(* Logix 5000 project; controller BTS01 vendor 1 type 14 code 217 rev 32.14; software revision 32.04; part 10 of 15 *)
(* tags used below, declared in another part *)
   Alarm_Active : DINT;
   Alarm_TMR : TIMER[17,32];
   ALM_ENABLE : DINT[25];
   GlobalAlmAck : BOOL;
   HMI_Alarms_Active : BOOL;
   HMI_Global_Alarm_Ack_PB : BOOL;
   HMIAlarms : DINT[25];   // Alarm Trigger Array
   HMIAlarmsMsg : STRING64[17,32];   // Alarm Descriptions to Match Alarm Trigger Array
(* Alarm, continued *)

ROUTINE Alarm_10   (* ladder *)
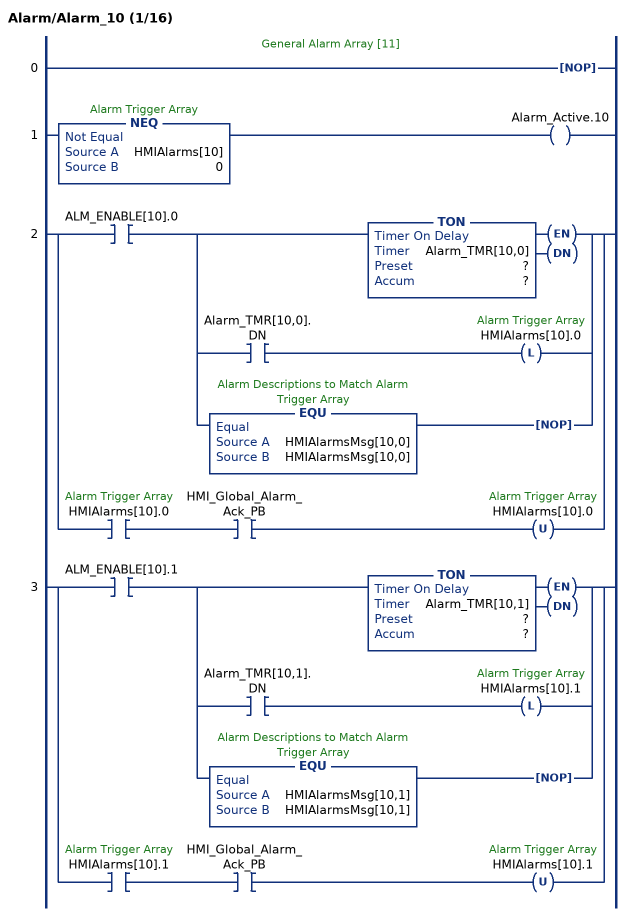
   // General Alarm Array [11]
   0: NOP();
   1: NEQ(HMIAlarms[10],0)OTE(Alarm_Active.10);
   2: [XIC(ALM_ENABLE[10].0) [TON(Alarm_TMR[10,0],?,?) ,XIC(Alarm_TMR[10,0].DN) OTL(HMIAlarms[10].0) ,EQU(HMIAlarmsMsg[10,0],HMIAlarmsMsg[10,0]) NOP() ] ,XIC(HMIAlarms[10].0) XIC(HMI_Global_Alarm_Ack_PB) OTU(HMIAlarms[10].0) ];
   3: [XIC(ALM_ENABLE[10].1) [TON(Alarm_TMR[10,1],?,?) ,XIC(Alarm_TMR[10,1].DN) OTL(HMIAlarms[10].1) ,EQU(HMIAlarmsMsg[10,1],HMIAlarmsMsg[10,1]) NOP() ] ,XIC(HMIAlarms[10].1) XIC(HMI_Global_Alarm_Ack_PB) OTU(HMIAlarms[10].1) ];
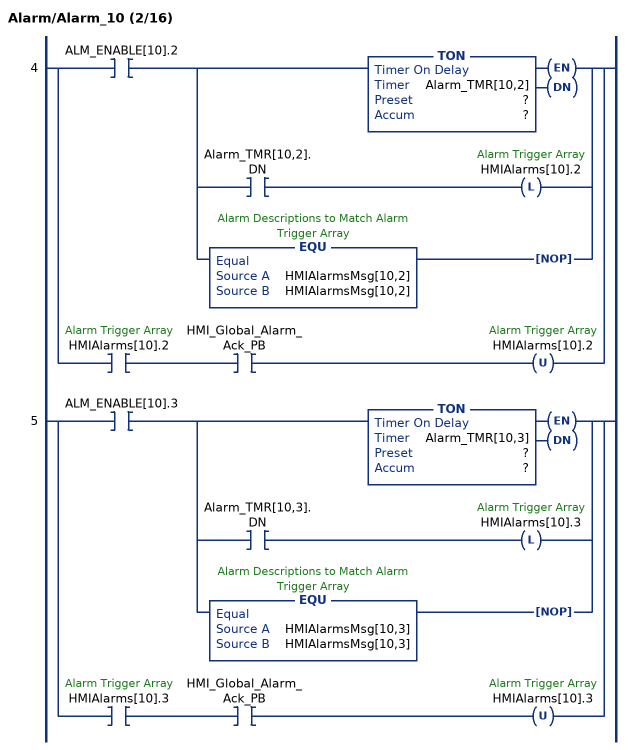
   4: [XIC(ALM_ENABLE[10].2) [TON(Alarm_TMR[10,2],?,?) ,XIC(Alarm_TMR[10,2].DN) OTL(HMIAlarms[10].2) ,EQU(HMIAlarmsMsg[10,2],HMIAlarmsMsg[10,2]) NOP() ] ,XIC(HMIAlarms[10].2) XIC(HMI_Global_Alarm_Ack_PB) OTU(HMIAlarms[10].2) ];
   5: [XIC(ALM_ENABLE[10].3) [TON(Alarm_TMR[10,3],?,?) ,XIC(Alarm_TMR[10,3].DN) OTL(HMIAlarms[10].3) ,EQU(HMIAlarmsMsg[10,3],HMIAlarmsMsg[10,3]) NOP() ] ,XIC(HMIAlarms[10].3) XIC(HMI_Global_Alarm_Ack_PB) OTU(HMIAlarms[10].3) ];
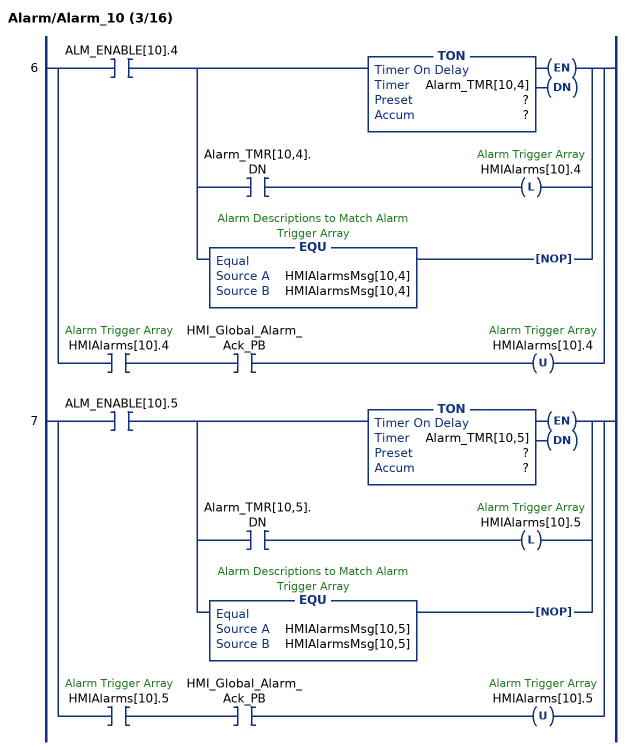
   6: [XIC(ALM_ENABLE[10].4) [TON(Alarm_TMR[10,4],?,?) ,XIC(Alarm_TMR[10,4].DN) OTL(HMIAlarms[10].4) ,EQU(HMIAlarmsMsg[10,4],HMIAlarmsMsg[10,4]) NOP() ] ,XIC(HMIAlarms[10].4) XIC(HMI_Global_Alarm_Ack_PB) OTU(HMIAlarms[10].4) ];
   7: [XIC(ALM_ENABLE[10].5) [TON(Alarm_TMR[10,5],?,?) ,XIC(Alarm_TMR[10,5].DN) OTL(HMIAlarms[10].5) ,EQU(HMIAlarmsMsg[10,5],HMIAlarmsMsg[10,5]) NOP() ] ,XIC(HMIAlarms[10].5) XIC(HMI_Global_Alarm_Ack_PB) OTU(HMIAlarms[10].5) ];
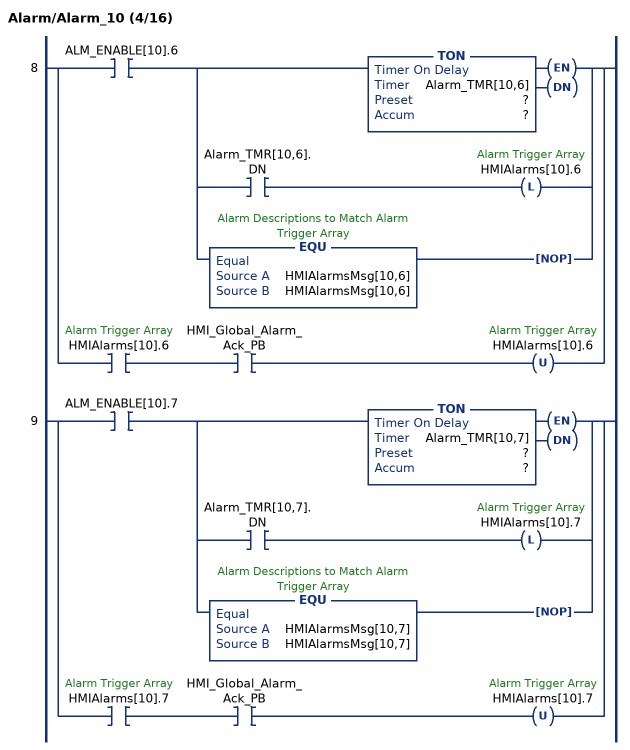
   8: [XIC(ALM_ENABLE[10].6) [TON(Alarm_TMR[10,6],?,?) ,XIC(Alarm_TMR[10,6].DN) OTL(HMIAlarms[10].6) ,EQU(HMIAlarmsMsg[10,6],HMIAlarmsMsg[10,6]) NOP() ] ,XIC(HMIAlarms[10].6) XIC(HMI_Global_Alarm_Ack_PB) OTU(HMIAlarms[10].6) ];
   9: [XIC(ALM_ENABLE[10].7) [TON(Alarm_TMR[10,7],?,?) ,XIC(Alarm_TMR[10,7].DN) OTL(HMIAlarms[10].7) ,EQU(HMIAlarmsMsg[10,7],HMIAlarmsMsg[10,7]) NOP() ] ,XIC(HMIAlarms[10].7) XIC(HMI_Global_Alarm_Ack_PB) OTU(HMIAlarms[10].7) ];
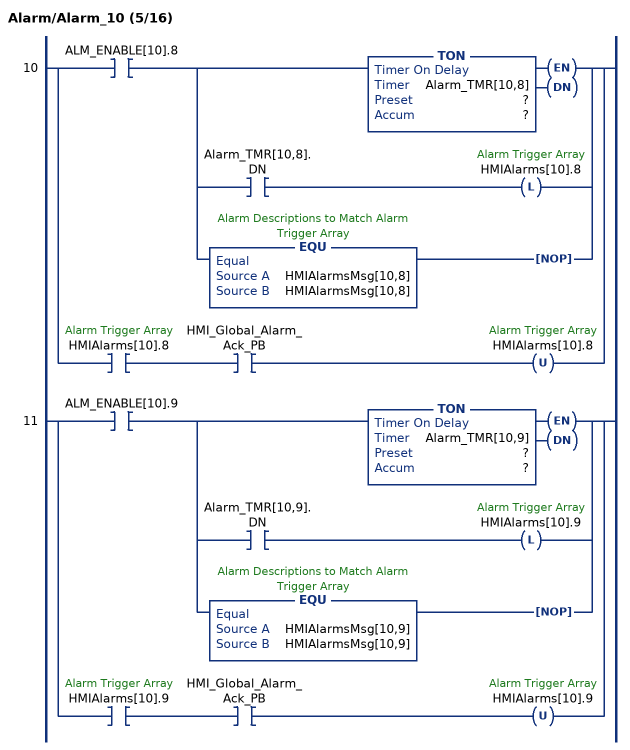
   10: [XIC(ALM_ENABLE[10].8) [TON(Alarm_TMR[10,8],?,?) ,XIC(Alarm_TMR[10,8].DN) OTL(HMIAlarms[10].8) ,EQU(HMIAlarmsMsg[10,8],HMIAlarmsMsg[10,8]) NOP() ] ,XIC(HMIAlarms[10].8) XIC(HMI_Global_Alarm_Ack_PB) OTU(HMIAlarms[10].8) ];
   11: [XIC(ALM_ENABLE[10].9) [TON(Alarm_TMR[10,9],?,?) ,XIC(Alarm_TMR[10,9].DN) OTL(HMIAlarms[10].9) ,EQU(HMIAlarmsMsg[10,9],HMIAlarmsMsg[10,9]) NOP() ] ,XIC(HMIAlarms[10].9) XIC(HMI_Global_Alarm_Ack_PB) OTU(HMIAlarms[10].9) ];
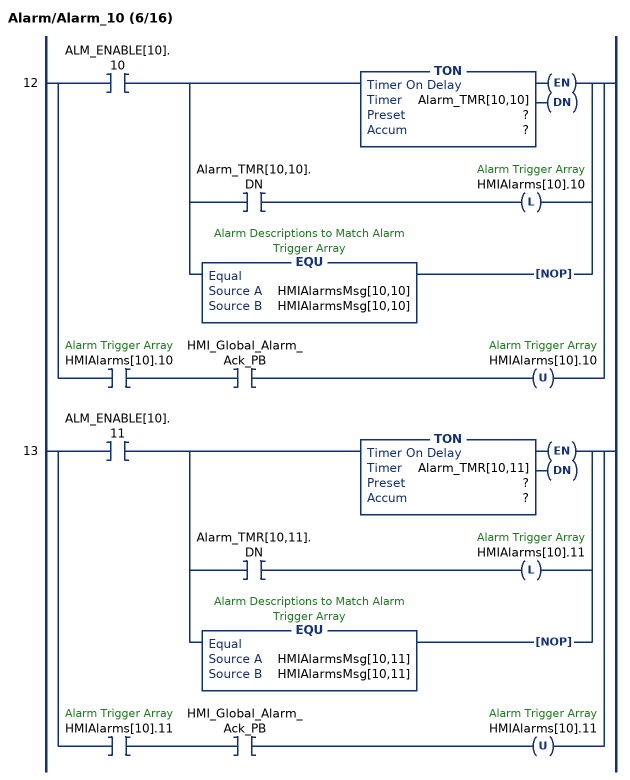
   12: [XIC(ALM_ENABLE[10].10) [TON(Alarm_TMR[10,10],?,?) ,XIC(Alarm_TMR[10,10].DN) OTL(HMIAlarms[10].10) ,EQU(HMIAlarmsMsg[10,10],HMIAlarmsMsg[10,10]) NOP() ] ,XIC(HMIAlarms[10].10) XIC(HMI_Global_Alarm_Ack_PB) OTU(HMIAlarms[10].10) ];
   13: [XIC(ALM_ENABLE[10].11) [TON(Alarm_TMR[10,11],?,?) ,XIC(Alarm_TMR[10,11].DN) OTL(HMIAlarms[10].11) ,EQU(HMIAlarmsMsg[10,11],HMIAlarmsMsg[10,11]) NOP() ] ,XIC(HMIAlarms[10].11) XIC(HMI_Global_Alarm_Ack_PB) OTU(HMIAlarms[10].11) ];
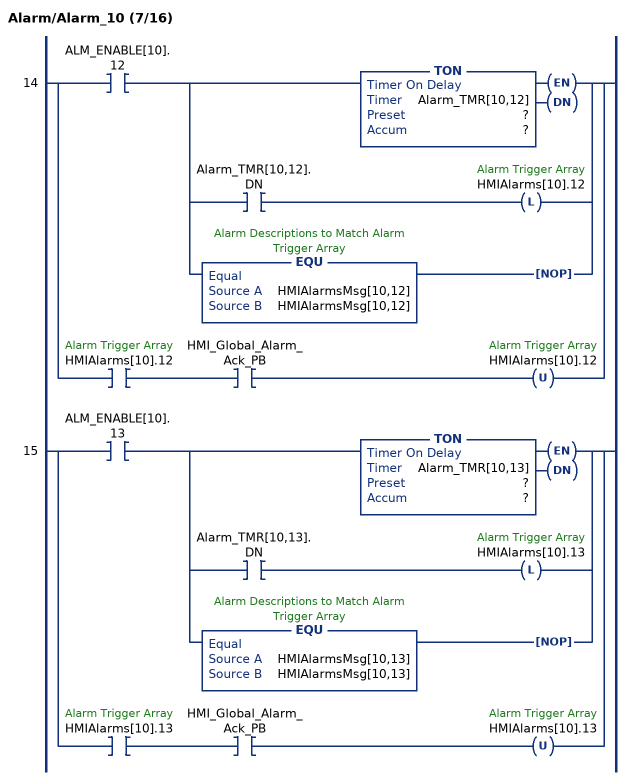
   14: [XIC(ALM_ENABLE[10].12) [TON(Alarm_TMR[10,12],?,?) ,XIC(Alarm_TMR[10,12].DN) OTL(HMIAlarms[10].12) ,EQU(HMIAlarmsMsg[10,12],HMIAlarmsMsg[10,12]) NOP() ] ,XIC(HMIAlarms[10].12) XIC(HMI_Global_Alarm_Ack_PB) OTU(HMIAlarms[10].12) ];
   15: [XIC(ALM_ENABLE[10].13) [TON(Alarm_TMR[10,13],?,?) ,XIC(Alarm_TMR[10,13].DN) OTL(HMIAlarms[10].13) ,EQU(HMIAlarmsMsg[10,13],HMIAlarmsMsg[10,13]) NOP() ] ,XIC(HMIAlarms[10].13) XIC(HMI_Global_Alarm_Ack_PB) OTU(HMIAlarms[10].13) ];
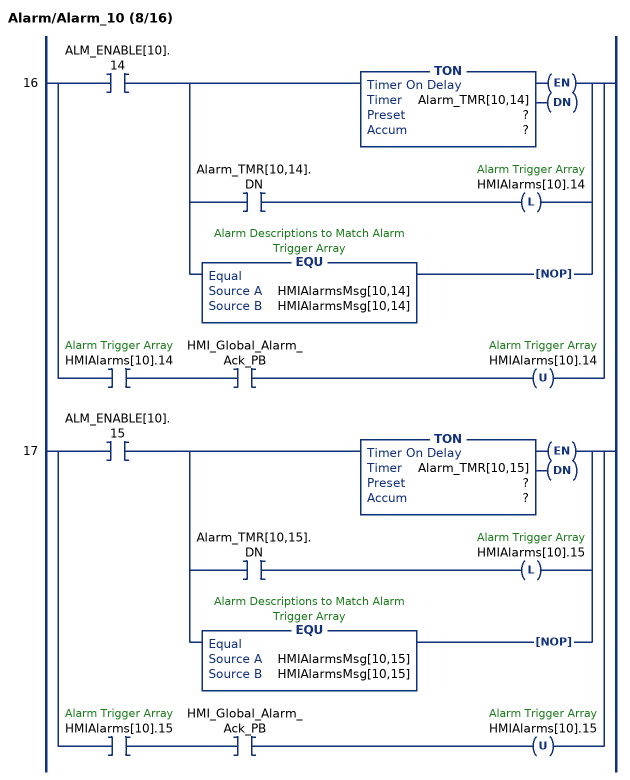
   16: [XIC(ALM_ENABLE[10].14) [TON(Alarm_TMR[10,14],?,?) ,XIC(Alarm_TMR[10,14].DN) OTL(HMIAlarms[10].14) ,EQU(HMIAlarmsMsg[10,14],HMIAlarmsMsg[10,14]) NOP() ] ,XIC(HMIAlarms[10].14) XIC(HMI_Global_Alarm_Ack_PB) OTU(HMIAlarms[10].14) ];
   17: [XIC(ALM_ENABLE[10].15) [TON(Alarm_TMR[10,15],?,?) ,XIC(Alarm_TMR[10,15].DN) OTL(HMIAlarms[10].15) ,EQU(HMIAlarmsMsg[10,15],HMIAlarmsMsg[10,15]) NOP() ] ,XIC(HMIAlarms[10].15) XIC(HMI_Global_Alarm_Ack_PB) OTU(HMIAlarms[10].15) ];
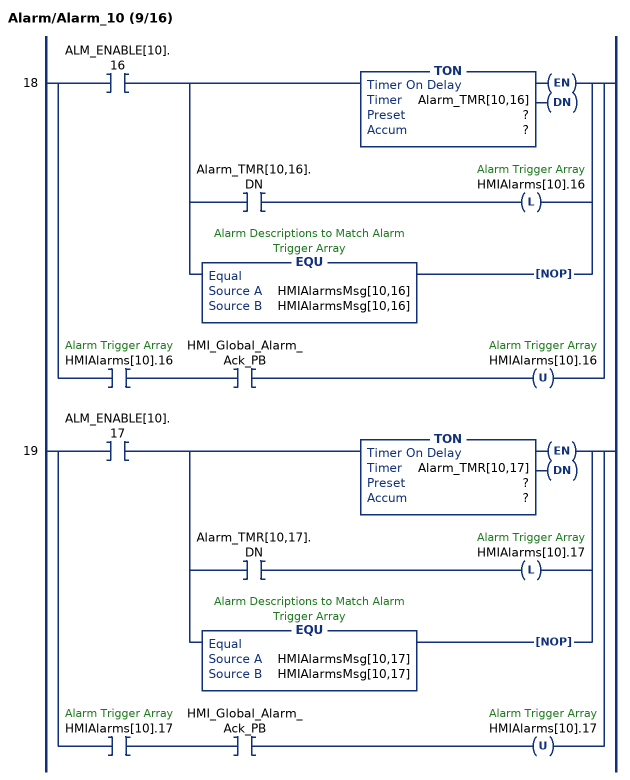
   18: [XIC(ALM_ENABLE[10].16) [TON(Alarm_TMR[10,16],?,?) ,XIC(Alarm_TMR[10,16].DN) OTL(HMIAlarms[10].16) ,EQU(HMIAlarmsMsg[10,16],HMIAlarmsMsg[10,16]) NOP() ] ,XIC(HMIAlarms[10].16) XIC(HMI_Global_Alarm_Ack_PB) OTU(HMIAlarms[10].16) ];
   19: [XIC(ALM_ENABLE[10].17) [TON(Alarm_TMR[10,17],?,?) ,XIC(Alarm_TMR[10,17].DN) OTL(HMIAlarms[10].17) ,EQU(HMIAlarmsMsg[10,17],HMIAlarmsMsg[10,17]) NOP() ] ,XIC(HMIAlarms[10].17) XIC(HMI_Global_Alarm_Ack_PB) OTU(HMIAlarms[10].17) ];
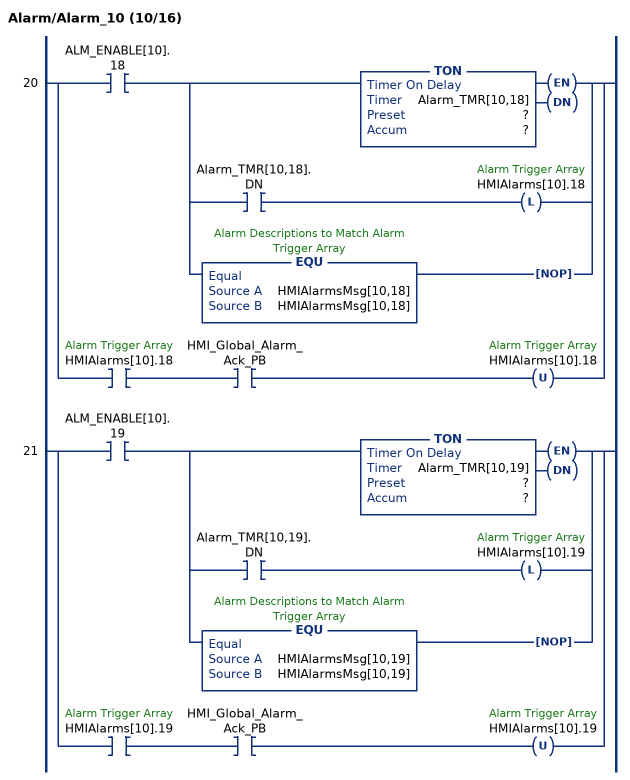
   20: [XIC(ALM_ENABLE[10].18) [TON(Alarm_TMR[10,18],?,?) ,XIC(Alarm_TMR[10,18].DN) OTL(HMIAlarms[10].18) ,EQU(HMIAlarmsMsg[10,18],HMIAlarmsMsg[10,18]) NOP() ] ,XIC(HMIAlarms[10].18) XIC(HMI_Global_Alarm_Ack_PB) OTU(HMIAlarms[10].18) ];
   21: [XIC(ALM_ENABLE[10].19) [TON(Alarm_TMR[10,19],?,?) ,XIC(Alarm_TMR[10,19].DN) OTL(HMIAlarms[10].19) ,EQU(HMIAlarmsMsg[10,19],HMIAlarmsMsg[10,19]) NOP() ] ,XIC(HMIAlarms[10].19) XIC(HMI_Global_Alarm_Ack_PB) OTU(HMIAlarms[10].19) ];
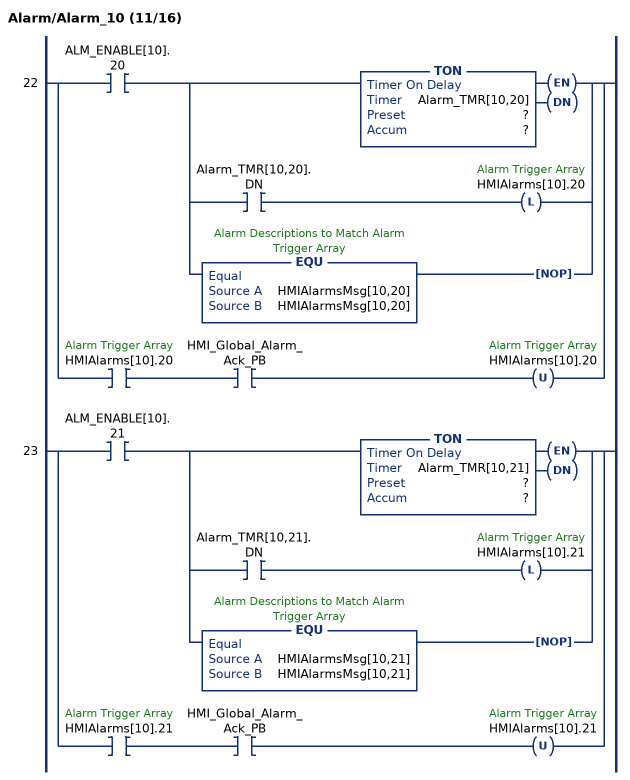
   22: [XIC(ALM_ENABLE[10].20) [TON(Alarm_TMR[10,20],?,?) ,XIC(Alarm_TMR[10,20].DN) OTL(HMIAlarms[10].20) ,EQU(HMIAlarmsMsg[10,20],HMIAlarmsMsg[10,20]) NOP() ] ,XIC(HMIAlarms[10].20) XIC(HMI_Global_Alarm_Ack_PB) OTU(HMIAlarms[10].20) ];
   23: [XIC(ALM_ENABLE[10].21) [TON(Alarm_TMR[10,21],?,?) ,XIC(Alarm_TMR[10,21].DN) OTL(HMIAlarms[10].21) ,EQU(HMIAlarmsMsg[10,21],HMIAlarmsMsg[10,21]) NOP() ] ,XIC(HMIAlarms[10].21) XIC(HMI_Global_Alarm_Ack_PB) OTU(HMIAlarms[10].21) ];
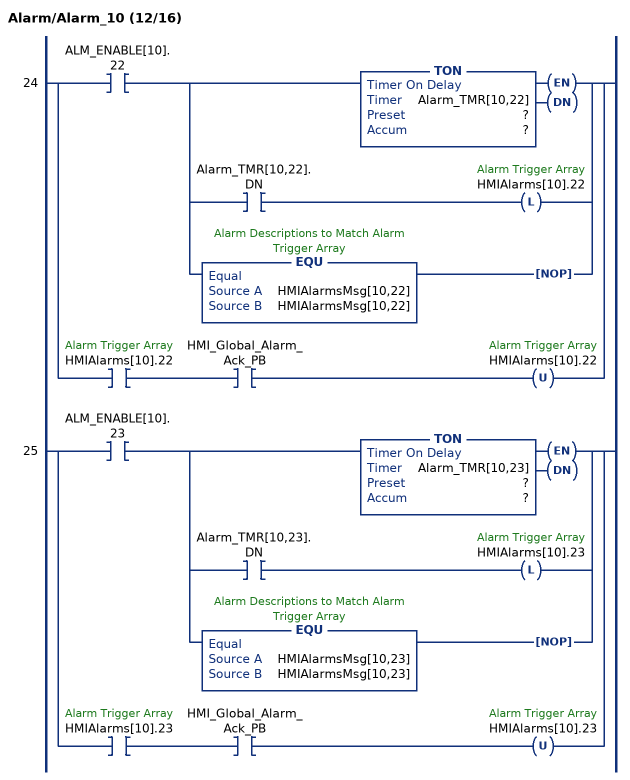
   24: [XIC(ALM_ENABLE[10].22) [TON(Alarm_TMR[10,22],?,?) ,XIC(Alarm_TMR[10,22].DN) OTL(HMIAlarms[10].22) ,EQU(HMIAlarmsMsg[10,22],HMIAlarmsMsg[10,22]) NOP() ] ,XIC(HMIAlarms[10].22) XIC(HMI_Global_Alarm_Ack_PB) OTU(HMIAlarms[10].22) ];
   25: [XIC(ALM_ENABLE[10].23) [TON(Alarm_TMR[10,23],?,?) ,XIC(Alarm_TMR[10,23].DN) OTL(HMIAlarms[10].23) ,EQU(HMIAlarmsMsg[10,23],HMIAlarmsMsg[10,23]) NOP() ] ,XIC(HMIAlarms[10].23) XIC(HMI_Global_Alarm_Ack_PB) OTU(HMIAlarms[10].23) ];
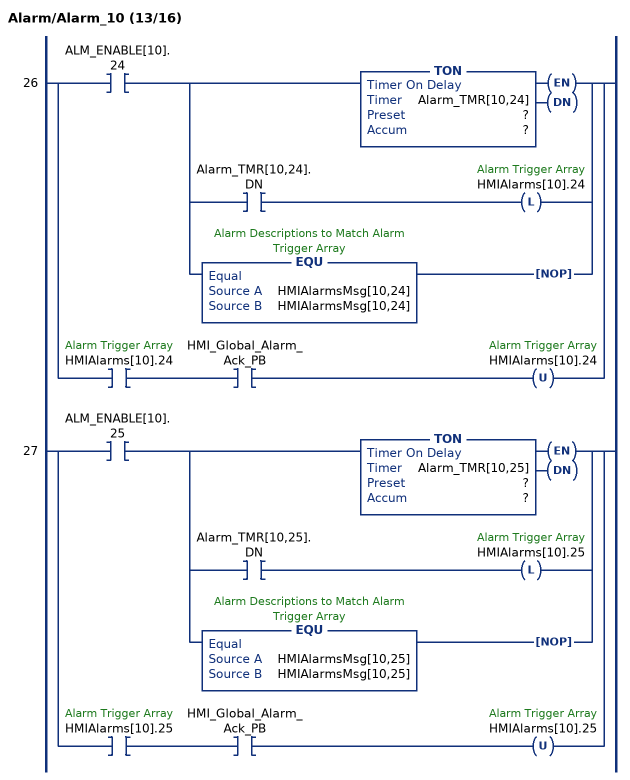
   26: [XIC(ALM_ENABLE[10].24) [TON(Alarm_TMR[10,24],?,?) ,XIC(Alarm_TMR[10,24].DN) OTL(HMIAlarms[10].24) ,EQU(HMIAlarmsMsg[10,24],HMIAlarmsMsg[10,24]) NOP() ] ,XIC(HMIAlarms[10].24) XIC(HMI_Global_Alarm_Ack_PB) OTU(HMIAlarms[10].24) ];
   27: [XIC(ALM_ENABLE[10].25) [TON(Alarm_TMR[10,25],?,?) ,XIC(Alarm_TMR[10,25].DN) OTL(HMIAlarms[10].25) ,EQU(HMIAlarmsMsg[10,25],HMIAlarmsMsg[10,25]) NOP() ] ,XIC(HMIAlarms[10].25) XIC(HMI_Global_Alarm_Ack_PB) OTU(HMIAlarms[10].25) ];
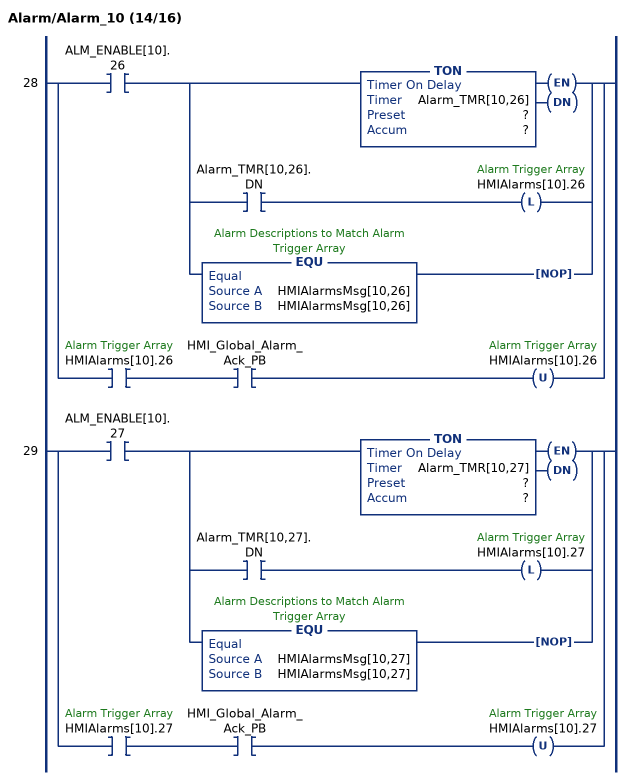
   28: [XIC(ALM_ENABLE[10].26) [TON(Alarm_TMR[10,26],?,?) ,XIC(Alarm_TMR[10,26].DN) OTL(HMIAlarms[10].26) ,EQU(HMIAlarmsMsg[10,26],HMIAlarmsMsg[10,26]) NOP() ] ,XIC(HMIAlarms[10].26) XIC(HMI_Global_Alarm_Ack_PB) OTU(HMIAlarms[10].26) ];
   29: [XIC(ALM_ENABLE[10].27) [TON(Alarm_TMR[10,27],?,?) ,XIC(Alarm_TMR[10,27].DN) OTL(HMIAlarms[10].27) ,EQU(HMIAlarmsMsg[10,27],HMIAlarmsMsg[10,27]) NOP() ] ,XIC(HMIAlarms[10].27) XIC(HMI_Global_Alarm_Ack_PB) OTU(HMIAlarms[10].27) ];
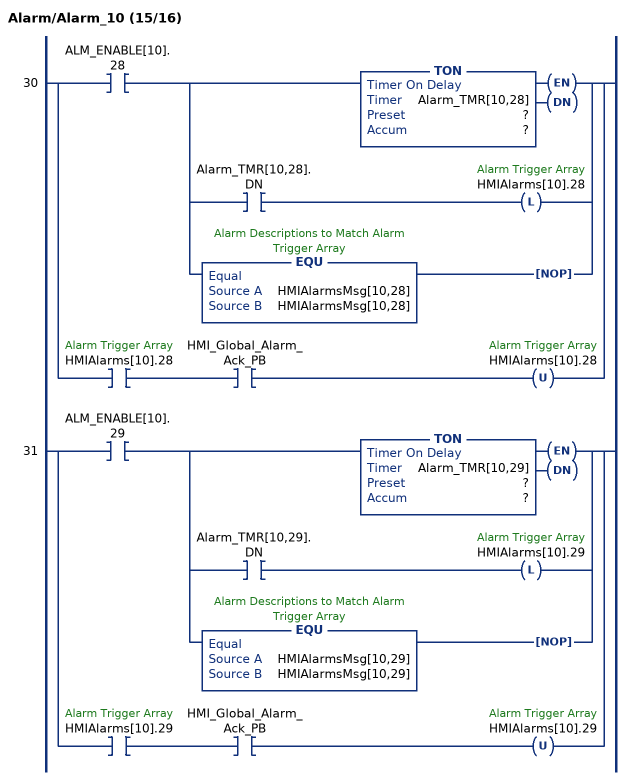
   30: [XIC(ALM_ENABLE[10].28) [TON(Alarm_TMR[10,28],?,?) ,XIC(Alarm_TMR[10,28].DN) OTL(HMIAlarms[10].28) ,EQU(HMIAlarmsMsg[10,28],HMIAlarmsMsg[10,28]) NOP() ] ,XIC(HMIAlarms[10].28) XIC(HMI_Global_Alarm_Ack_PB) OTU(HMIAlarms[10].28) ];
   31: [XIC(ALM_ENABLE[10].29) [TON(Alarm_TMR[10,29],?,?) ,XIC(Alarm_TMR[10,29].DN) OTL(HMIAlarms[10].29) ,EQU(HMIAlarmsMsg[10,29],HMIAlarmsMsg[10,29]) NOP() ] ,XIC(HMIAlarms[10].29) XIC(HMI_Global_Alarm_Ack_PB) OTU(HMIAlarms[10].29) ];
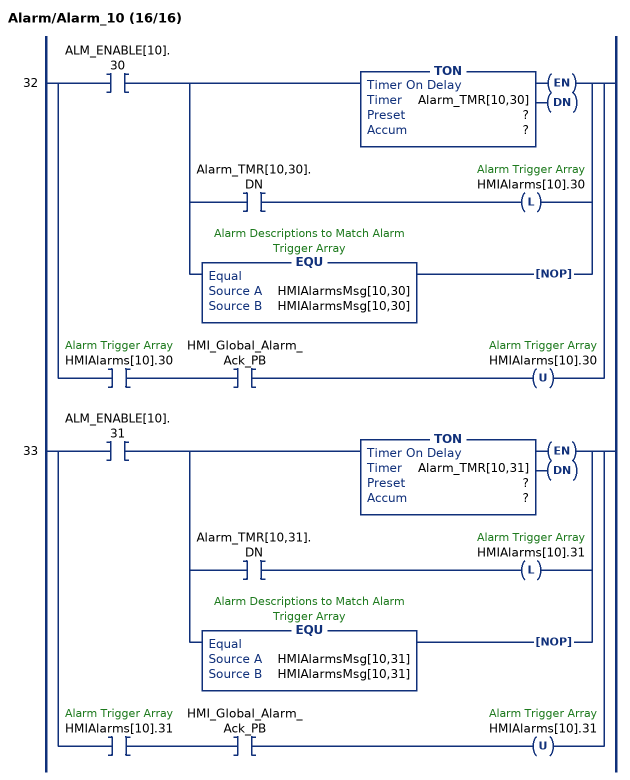
   32: [XIC(ALM_ENABLE[10].30) [TON(Alarm_TMR[10,30],?,?) ,XIC(Alarm_TMR[10,30].DN) OTL(HMIAlarms[10].30) ,EQU(HMIAlarmsMsg[10,30],HMIAlarmsMsg[10,30]) NOP() ] ,XIC(HMIAlarms[10].30) XIC(HMI_Global_Alarm_Ack_PB) OTU(HMIAlarms[10].30) ];
   33: [XIC(ALM_ENABLE[10].31) [TON(Alarm_TMR[10,31],?,?) ,XIC(Alarm_TMR[10,31].DN) OTL(HMIAlarms[10].31) ,EQU(HMIAlarmsMsg[10,31],HMIAlarmsMsg[10,31]) NOP() ] ,XIC(HMIAlarms[10].31) XIC(HMI_Global_Alarm_Ack_PB) OTU(HMIAlarms[10].31) ];
END_ROUTINE

ROUTINE Alarm_Main   (* ladder *)
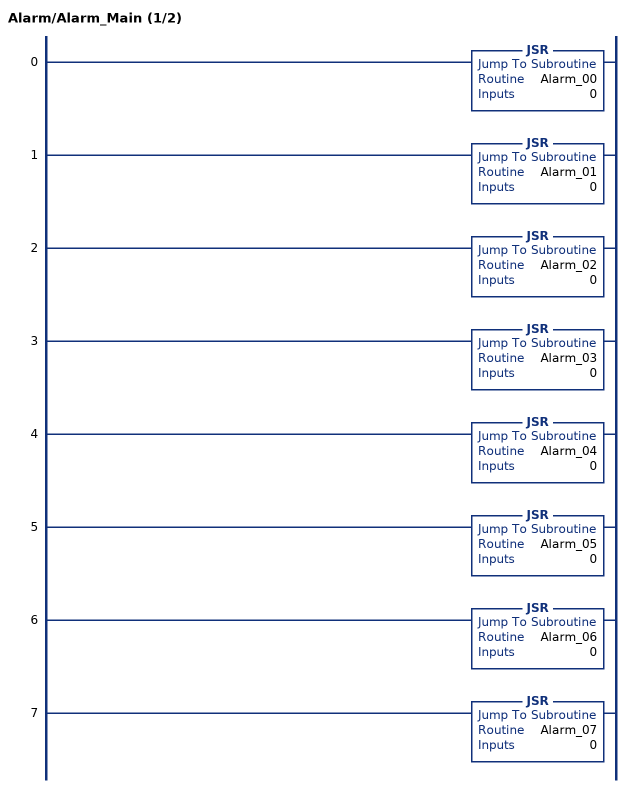
   0: JSR(Alarm_00,0);
   1: JSR(Alarm_01,0);
   2: JSR(Alarm_02,0);
   3: JSR(Alarm_03,0);
   4: JSR(Alarm_04,0);
   5: JSR(Alarm_05,0);
   6: JSR(Alarm_06,0);
   7: JSR(Alarm_07,0);
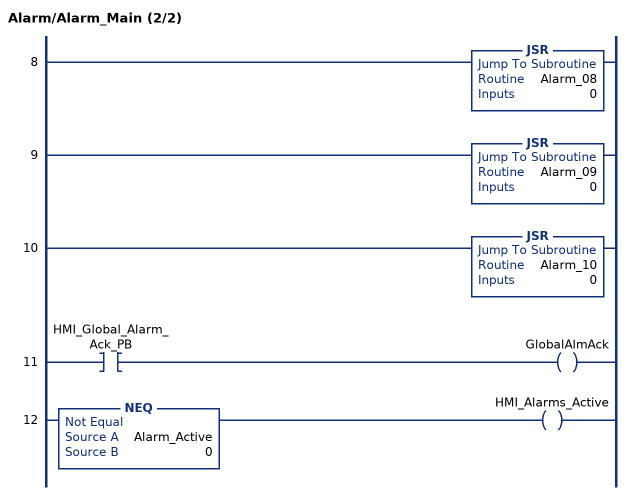
   8: JSR(Alarm_08,0);
   9: JSR(Alarm_09,0);
   10: JSR(Alarm_10,0);
   11: XIC(HMI_Global_Alarm_Ack_PB)OTE(GlobalAlmAck);
   12: NEQ(Alarm_Active,0)OTE(HMI_Alarms_Active);
END_ROUTINE
END_PROGRAM
